# EPICS autosave request: ADmarCCD/marCCDApp/Db/marCCD_settings.req
$(P)$(R)ReadTiffTimeout
$(P)$(R)OverlapMode
$(P)$(R)AutoSave
$(P)$(R)FrameShift
$(P)$(R)Stability
$(P)$(R)DetectorDistance
$(P)$(R)BeamX
$(P)$(R)BeamY
$(P)$(R)StartPhi
$(P)$(R)RotationAxis
$(P)$(R)RotationRange
$(P)$(R)TwoTheta
$(P)$(R)Wavelength
$(P)$(R)FileComments
$(P)$(R)DatasetComments
$(P)$(R)GateMode
$(P)$(R)ReadoutMode
$(P)$(R)SeriesFileTemplate
$(P)$(R)SeriesFileDigits
$(P)$(R)SeriesFileFirst
